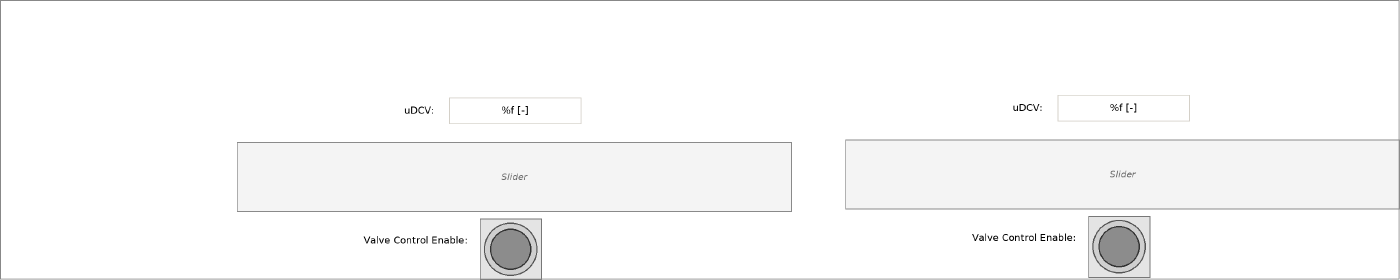
VISUALIZATION Visualization  // 1590x319
    Slider (269,162 630x79), variable: Inputs.uDcvMainJib, scale -1..1
    PushSwitchLed (545,249 70x70), variable: Inputs.uDcvEnableMainJib, behaviour: TOGGLE, style: Switch-PushSwitchLed-Gray
    Textfield (510,111 150x30), "%f [-]", text variable: Inputs.uDcvMainJib
        OnMouseClick: write the text variable via Default, min -1, max 1
    Label (443,111 66x30), "uDCV:"
    Label (381,259 182x30), "Valve Control Enable:"
    Slider (960,159 630x79), variable: Inputs.uDcvKnuckleJib, scale -1..1
    PushSwitchLed (1236,246 70x70), variable: Inputs.uDcvEnableKnuckleJib, behaviour: TOGGLE, style: Switch-PushSwitchLed-Gray
    Textfield (1201,108 150x30), "%f [-]", text variable: Inputs.uDcvKnuckleJib
        OnMouseClick: write the text variable via Default, min -1, max 1
    Label (1134,108 66x30), "uDCV:"
    Label (1072,256 182x30), "Valve Control Enable:"
END_VISUALIZATION

(* stored: Version 1.1.0.1, ProductVersion 3.1.4024.9
   Visu Visualization: Id {d8dee94c-064f-4243-8341-9a26801948ea} *)
